FUNCTION_BLOCK Sequence5
VAR_INPUT
END_VAR
VAR_OUTPUT
END_VAR
VAR
END_VAR

END_FUNCTION_BLOCK

(* stored: Version 1.1.0.1, ProductVersion 3.1.4024.11
   POU Sequence5: Id {fa7ef538-1527-401e-8789-806f3b39bcb1}, SpecialFunc None *)
